# EPICS autosave request: iocBoot/iocvxWorks/auto_positions.req
$(P)m1.OFF
$(P)m1.DVAL
$(P)m2.OFF
$(P)m2.DVAL
$(P)m3.OFF
$(P)m3.DVAL
$(P)m4.OFF
$(P)m4.DVAL
$(P)m5.OFF
$(P)m5.DVAL
$(P)m6.OFF
$(P)m6.DVAL
$(P)m7.OFF
$(P)m7.DVAL
$(P)m8.OFF
$(P)m8.DVAL
$(P)m9.OFF
$(P)m9.DVAL
$(P)m10.OFF
$(P)m10.DVAL
$(P)m11.OFF
$(P)m11.DVAL
$(P)m12.OFF
$(P)m12.DVAL
$(P)m13.OFF
$(P)m13.DVAL
$(P)m14.OFF
$(P)m14.DVAL
$(P)m15.OFF
$(P)m15.DVAL
$(P)m16.OFF
$(P)m16.DVAL
